Universal Robots PolyScope program: 0609.urp

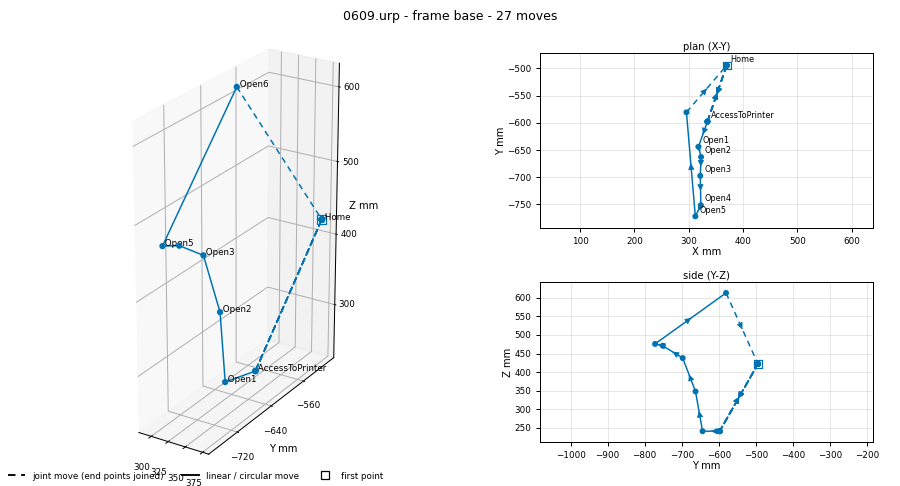
[picture p0: tool path of 0609.urp in frame base, 27 of 27 moves have a stored position in this frame; points joined in program order, loops and branches not executed]
Program 0609 (installation=default directory=/programs/usbdisk/새로운 폴더_2 createdIn=5.12.7.1102192 lastSavedIn=5.11.0.108249 robotSerialNumber=20215501208)
Calibrated DH parameters: a=[0.000135, -0.201821, -0.391913, -0.000063, 0.000038, 0]; d=[0.162484, -479.507804, 481.562221, -1.92078, 0.099549, 0.099572]; alpha=[1.570789, -0.00078, 0.007148, 1.569147, -1.569841, 0]; deltaTheta=[0, 1.075971, -1.038513, -0.037456, 0, 0]
Robot Program (runOnlyOnce=false)
  Folder Init
    Call Init_Variables
    Call Socket_Open
    MoveJ speed 60 deg/s, acceleration 80 deg/s^2 (useActiveTCP=true) feature=Base
      Waypoint Home: TCP in base x=369.65 y=-494.569 z=421.925 mm, rx=0.0496 ry=-3.0772 rz=-0.0574 rad; joints [-245.337, -73.512, 79.652, 267.34, -92.102, 23.034] deg
  Folder Main Sequence
    Folder Task1:OpenPrinter
      Call Enter_Next_Task
      Loop While (checkContinuously=false) expression=retry_count <= max_retry and task_done == 0
        MoveJ speed 60 deg/s, acceleration 80 deg/s^2 (useActiveTCP=true) feature=Base
          Waypoint Home: TCP in base x=369.65 y=-494.569 z=421.925 mm, rx=0.0496 ry=-3.0772 rz=-0.0574 rad; joints [-245.337, -73.512, 79.652, 267.34, -92.102, 23.034] deg
          Waypoint AccessToPrinter: TCP in base x=334.462 y=-597.737 z=240.467 mm, rx=-0.0069 ry=3.1388 rz=-0.0445 rad; joints [-252.013, -58.111, 86.313, 240.264, -90.06, 18.038] deg
          MoveL speed 250 mm/s, acceleration 1200 mm/s^2 (useActiveTCP=true) feature=Base
            Waypoint Open1: TCP in base x=318.021 y=-643.967 z=240.481 mm, rx=-0.0068 ry=3.1388 rz=-0.0445 rad; joints [-254.436, -54.011, 79.432, 243.032, -89.985, 15.598] deg
            Waypoint Open2: TCP in base x=322.784 y=-662.887 z=347.649 mm, rx=0.0033 ry=-3.1272 rz=-0.039 rad; joints [-254.437, -55.388, 64.401, 262.634, -90.038, 15.606] deg
            Waypoint Open3: TCP in base x=321.329 y=-697.509 z=437.722 mm, rx=0.0214 ry=3.1194 rz=-0.1204 rad; joints [-255.276, -52.597, 48.232, 269.856, -89.693, 15.609] deg
            Waypoint Open4: TCP in base x=322.369 y=-751.555 z=471.14 mm, rx=-0.056 ry=3.0495 rz=-0.4423 rad; joints [-256.148, -45.626, 35.019, 263.813, -89.938, 11.834] deg
            Waypoint Open5: TCP in base x=312.24 y=-772.06 z=475.94 mm, rx=-0.0354 ry=3.0161 rz=-0.6648 rad; joints [-256.943, -44.398, 34.822, 254.694, -91.917, 11.398] deg
            Waypoint Open6: TCP in base x=295.845 y=-580.619 z=613.456 mm, rx=-0.0405 ry=-3.057 rz=-0.0586 rad; joints [-254.175, -62.295, 34.865, 300.956, -93.656, 17.369] deg
        Call Check_Door_Open
        Switch expression=fail_flag
          Case (caseValue=0)
            Script: task_done = 1
          Case (caseValue=1)
            Script: retry_count = retry_count + 1
      If task_done == 0
        Call Error_Stop
    Folder Task2:PickA4FromTray
      Call Enter_Next_Task
      MoveJ speed 60 deg/s, acceleration 80 deg/s^2 (useActiveTCP=true) feature=Base
        Waypoint Home: TCP in base x=369.65 y=-494.569 z=421.925 mm, rx=0.0496 ry=-3.0772 rz=-0.0574 rad; joints [-245.337, -73.512, 79.652, 267.34, -92.102, 23.034] deg
        Waypoint AccessToTray: TCP in base x=369.603 y=-494.616 z=422.071 mm, rx=0.0496 ry=-3.0774 rz=-0.0569 rad; joints [-245.343, -73.517, 79.642, 267.335, -92.098, 23.025] deg
      Call Gripper_Open
      Call Wait_Motor_Idle
      Call DC_Run
      Call Wait_Motor_Idle
      Call Gripper_Close
      Call Wait_Motor_Idle
      MoveJ speed 60 deg/s, acceleration 80 deg/s^2 (useActiveTCP=true) feature=Base
        Waypoint RetreatFromTray: TCP in base x=369.611 y=-494.615 z=422.061 mm, rx=0.0496 ry=-3.0774 rz=-0.057 rad; joints [-245.343, -73.516, 79.642, 267.335, -92.097, 23.027] deg
      If fail_flag == 1
        Call Error_Stop
    Folder Task3:PlaceA4OnScanner
      Call Enter_Next_Task
      MoveJ speed 60 deg/s, acceleration 80 deg/s^2 (useActiveTCP=true) feature=Base
        Waypoint AccessToScanne: TCP in base x=369.631 y=-494.591 z=421.924 mm, rx=0.0495 ry=-3.0773 rz=-0.0574 rad; joints [-245.34, -73.511, 79.65, 267.341, -92.099, 23.034] deg
      Call Gripper_Open
      Call Wait_Motor_Idle
      MoveJ speed 60 deg/s, acceleration 80 deg/s^2 (useActiveTCP=true) feature=Base
        Waypoint RetreatFromScan: TCP in base x=369.639 y=-494.607 z=421.869 mm, rx=0.0495 ry=-3.0772 rz=-0.0575 rad; joints [-245.339, -73.506, 79.652, 267.339, -92.104, 23.035] deg
      Call Check_Paper_Detected
      If fail_flag == 1
        Call Error_Stop
    Folder Task4:ClosePrinter
      Call Enter_Next_Task
      Loop While (checkContinuously=false) expression=retry_count <= max_retry and task_done == 0
        MoveJ speed 60 deg/s, acceleration 80 deg/s^2 (useActiveTCP=true) feature=Base
          Waypoint AccessToPrinter: TCP in base x=334.462 y=-597.737 z=240.467 mm, rx=-0.0069 ry=3.1388 rz=-0.0445 rad; joints [-252.013, -58.111, 86.313, 240.264, -90.06, 18.038] deg
          Waypoint ClosePrinterr: TCP in base x=369.641 y=-494.609 z=421.879 mm, rx=0.0495 ry=-3.0772 rz=-0.0575 rad; joints [-245.339, -73.506, 79.651, 267.339, -92.101, 23.035] deg
          Waypoint RetreatFromPrin: TCP in base x=369.644 y=-494.592 z=421.887 mm, rx=0.0495 ry=-3.0772 rz=-0.0574 rad; joints [-245.338, -73.509, 79.653, 267.337, -92.102, 23.034] deg
        Call Check_Door_Closed
        Switch expression=fail_flag
          Case (caseValue=0)
            Script: task_done = 1
          Case (caseValue=1)
            Script: retry_count = retry_count + 1
      If task_done == 0
        Call Error_Stop
    Folder Task5:OpenPrinter
      Call Enter_Next_Task
      Loop While (checkContinuously=false) expression=retry_count <= max_retry and task_done == 0
        MoveJ speed 60 deg/s, acceleration 80 deg/s^2 (useActiveTCP=true) feature=Base
          Waypoint AccessToPrinter: TCP in base x=334.462 y=-597.737 z=240.467 mm, rx=-0.0069 ry=3.1388 rz=-0.0445 rad; joints [-252.013, -58.111, 86.313, 240.264, -90.06, 18.038] deg
          Waypoint OpenPrinterr: TCP in base x=369.668 y=-494.585 z=421.902 mm, rx=0.0496 ry=-3.0772 rz=-0.0574 rad; joints [-245.336, -73.508, 79.649, 267.341, -92.102, 23.034] deg
          Waypoint RetreatFromPrin: TCP in base x=369.644 y=-494.592 z=421.887 mm, rx=0.0495 ry=-3.0772 rz=-0.0574 rad; joints [-245.338, -73.509, 79.653, 267.337, -92.102, 23.034] deg
        Call Check_Door_Open
        Switch expression=fail_flag
          Case (caseValue=0)
            Script: task_done = 1
          Case (caseValue=1)
            Script: retry_count = retry_count + 1
      If task_done == 0
        Call Error_Stop
    Folder Task6:PickA4FromScanner
      Call Enter_Next_Task
      Call Gripper_Open
      Call Wait_Motor_Idle
      MoveJ speed 60 deg/s, acceleration 80 deg/s^2 (useActiveTCP=true) feature=Base
        Waypoint AccessToScanner: TCP in base x=369.655 y=-494.587 z=421.911 mm, rx=0.0495 ry=-3.0772 rz=-0.0574 rad; joints [-245.337, -73.508, 79.649, 267.341, -92.103, 23.036] deg
      Call Gripper_Close
      Call Wait_Motor_Idle
      MoveJ speed 60 deg/s, acceleration 80 deg/s^2 (useActiveTCP=true) feature=Base
        Waypoint RetreatFromSca: TCP in base x=369.664 y=-494.583 z=421.908 mm, rx=0.0496 ry=-3.0772 rz=-0.0574 rad; joints [-245.336, -73.508, 79.649, 267.341, -92.102, 23.034] deg
      If fail_flag == 1
        Call Error_Stop
    Folder Task7:PlaceA4InBasket
      Call Enter_Next_Task
      MoveJ speed 60 deg/s, acceleration 80 deg/s^2 (useActiveTCP=true) feature=Base
        Waypoint AccessToBasket: TCP in base x=369.638 y=-494.57 z=421.942 mm, rx=0.0496 ry=-3.0772 rz=-0.0573 rad; joints [-245.338, -73.513, 79.652, 267.339, -92.104, 23.032] deg
      Call Gripper_Open
      Call Wait_Motor_Idle
      MoveJ speed 60 deg/s, acceleration 80 deg/s^2 (useActiveTCP=true) feature=Base
        Waypoint RetreatFromBask: TCP in base x=369.654 y=-494.572 z=421.913 mm, rx=0.0496 ry=-3.0772 rz=-0.0574 rad; joints [-245.336, -73.511, 79.652, 267.339, -92.103, 23.033] deg
      If fail_flag == 1
        Call Error_Stop
    Folder Task8:ClosePrinter
      Call Enter_Next_Task
      Loop While (checkContinuously=false) expression=retry_count <= max_retry and task_done == 0
        MoveJ speed 60 deg/s, acceleration 80 deg/s^2 (useActiveTCP=true) feature=Base
          Waypoint AccessToPrinter: TCP in base x=334.462 y=-597.737 z=240.467 mm, rx=-0.0069 ry=3.1388 rz=-0.0445 rad; joints [-252.013, -58.111, 86.313, 240.264, -90.06, 18.038] deg
          Waypoint ClosePrinter: TCP in base x=369.674 y=-494.571 z=421.895 mm, rx=0.0496 ry=-3.0772 rz=-0.0574 rad; joints [-245.335, -73.508, 79.651, 267.341, -92.102, 23.034] deg
          Waypoint RetreatFromPrin: TCP in base x=369.644 y=-494.592 z=421.887 mm, rx=0.0495 ry=-3.0772 rz=-0.0574 rad; joints [-245.338, -73.509, 79.653, 267.337, -92.102, 23.034] deg
        Call Check_Door_Closed
        Switch expression=fail_flag
          Case (caseValue=0)
            Script: task_done = 1
          Case (caseValue=1)
            Script: retry_count = retry_count + 1
      If task_done == 0
        Call Error_Stop
SubProgram -> Socket_Open
SubProgram -> Init_Variables
SubProgram -> DC_Run
SubProgram -> Gripper_Close
SubProgram -> Gripper_Open
SubProgram -> Wait_Motor_Idle
SubProgram -> Check_Door_Closed
SubProgram -> Check_Door_Open
SubProgram -> Check_Paper_Detected
SubProgram -> Error_Stop
SubProgram -> Enter_Next_Task
SubProgram Init_Variables (keepSynchronizedWithDisk=false)
  Script file /programs/usbdisk/scripts/Init_Variables.script
    | # Retry / fail control
    | global retry_count = 0
    | global max_retry = 2
    | global fail_flag = 0
    | global task_done = 0
    | global current_task = 0
    | 
    | # State variables
    | global door_state = 0      # 0: closed, 1: open
    | global motor_state = 0     # 0: idle, 1: busy
    | global paper_state = 0     # 0: not detected, 1: detected
    | 
    | # Socket / response
    | global socket_state = False
    | global pc_response = ""
    | 
    | # ============================================================
    | # Command strings
    | # URScript → PC Server → Arduino
    | # ============================================================
    | 
    | global CMD_PING = "PING\n"
    | global CMD_GRIPPER_OPEN = "G OPEN\n"
    | global CMD_GRIPPER_CLOSE = "G CLOSE\n"
    | global CMD_DC_RUN = "D RUN\n"
    | global CMD_ESTOP = "ESTOP\n"
    | global CMD_MOTOR_STATUS = "MOTOR STATUS\n"
    | global CMD_DOOR_STATUS = "DOOR STATUS\n"
    | global CMD_CAMERA = "V CAMERA\n"
    | 
    | # ============================================================
    | # Expected response strings
    | # Arduino / PC Server → URScript
    | # ============================================================
    | 
    | global RESP_OK_PING = "OK PING"
    | global RESP_OK_GRIPPER_OPEN = "OK G OPEN"
    | global RESP_OK_GRIPPER_CLOSE = "OK G CLOSE"
    | global RESP_OK_DC_RUN = "OK D RUN"
    | global RESP_OK_ESTOP = "OK ESTOP"
    | 
    | global RESP_MOTOR_BUSY = "MOTOR STATUS BUSY"
    | global RESP_MOTOR_IDLE = "MOTOR STATUS IDLE"
    | 
    | global RESP_DOOR_OPEN = "DOOR STATUS OPEN"
    | global RESP_DOOR_CLOSED = "DOOR STATUS CLOSED"
    | 
    | global RESP_PAPER_DETECTED = "PAPER DETECTED"
    | global RESP_PAPER_NOT_DETECTED = "PAPER NOT DETECTED"
SubProgram Socket_Open (keepSynchronizedWithDisk=false)
  Script file /programs/usbdisk/scripts/Socket_Open.script
    | global socket_state = socket_open("192.168.0.10", 5000)
    | 
    | if socket_state:
    |   socket_send_string(CMD_PING)
    |   global pc_response = socket_read_line()
    | 
    |   if pc_response == RESP_OK_PING:
    |     global fail_flag = 0
    |     textmsg("Socket open OK")
    |   else:
    |     global fail_flag = 1
    |     textmsg("PING failed: ", pc_response)
    |   end
    | 
    | else:
    |   global fail_flag = 1
    |   textmsg("Socket open FAILED")
    |   halt
    | end
SubProgram Enter_Next_Task (keepSynchronizedWithDisk=false)
  Script file /programs/usbdisk/scripts/Enter_Next_Task.script
    | global current_task = current_task + 1
    | global retry_count = 0
    | global task_done = 0
    | global fail_flag = 0
SubProgram Check_Door_Open (keepSynchronizedWithDisk=false)
  Script file /programs/usbdisk/Check_Door_Open.script
    | socket_send_string(CMD_DOOR_STATUS)
    | global pc_response = socket_read_line()
    | 
    | if pc_response == RESP_DOOR_OPEN:
    |   global door_state = 1
    |   global fail_flag = 0
    | 
    | elif pc_response == RESP_DOOR_CLOSED:
    |   global door_state = 0
    |   global fail_flag = 1
    | 
    | else:
    |   global fail_flag = 1
    | end
SubProgram Error_Stop (keepSynchronizedWithDisk=false)
  Script file /programs/usbdisk/Error_Stop.script
    | # 현재 task 번호에 따라 오류 메시지 출력
    | if current_task == 1:
    |   popup("Task 1 Failed: Open Printer", title="Task Error", warning=True, error=False)
    | 
    | elif current_task == 2:
    |   popup("Task 2 Failed: Pick A4 From Paper Box", title="Task Error", warning=True, error=False)
    | 
    | elif current_task == 3:
    |   popup("Task 3 Failed: Place A4 To Printer Head", title="Task Error", warning=True, error=False)
    | 
    | elif current_task == 4:
    |   popup("Task 4 Failed: Close Printer", title="Task Error", warning=True, error=False)
    | 
    | elif current_task == 5:
    |   popup("Task 5 Failed: Open Printer Again", title="Task Error", warning=True, error=False)
    | 
    | elif current_task == 6:
    |   popup("Task 6 Failed: Pick A4 From Printer Head", title="Task Error", warning=True, error=False)
    | 
    | elif current_task == 7:
    |   popup("Task 7 Failed: Place A4 To Paper Box", title="Task Error", warning=True, error=False)
    | 
    | elif current_task == 8:
    |   popup("Task 8 Failed: Close Printer Again", title="Task Error", warning=True, error=False)
    | 
    | else:
    |   popup("Unknown Task Failed", title="Task Error", warning=True, error=False)
    | end
    | 
    | # Arduino/PC 측 정지 요청
    | socket_send_string(CMD_ESTOP)
    | global pc_response = socket_read_line()
    | 
    | # 로그 출력
    | textmsg("ESTOP response: ", pc_response)
    | 
    | # UR Program 정지
    | halt
SubProgram Gripper_Open (keepSynchronizedWithDisk=false)
  Script file /programs/usbdisk/Gripper_Open.script
    | socket_send_string(CMD_GRIPPER_OPEN)
    | global pc_response = socket_read_line()
    | 
    | if pc_response == RESP_OK_GRIPPER_OPEN:
    |   global motor_state = 1
    |   global fail_flag = 0
    | else:
    |   global fail_flag = 1
    | end
SubProgram Wait_Motor_Idle (keepSynchronizedWithDisk=false)
  Script file /programs/usbdisk/scripts/Wait_Motor_Idle.script
    | # MOTOR STATUS를 반복 조회하여 IDLE이 될 때까지 대기
    | # break문 사용 불가하므로 wait_done 임시 변수 사용
    | 
    | wait_done = 0
    | 
    | while wait_done == 0:
    |   socket_send_string(CMD_MOTOR_STATUS)
    |   global pc_response = socket_read_line()
    | 
    |   if pc_response == RESP_MOTOR_BUSY:
    |     global motor_state = 1
    |     sleep(0.1)
    | 
    |   elif pc_response == RESP_MOTOR_IDLE:
    |     global motor_state = 0
    |     global fail_flag = 0
    |     global wait_done = 1
    | 
    |   else:
    |     global fail_flag = 1
    |     global wait_done = 1
    |   end
    | end
SubProgram DC_Run (keepSynchronizedWithDisk=false)
  Script file /programs/usbdisk/DC_Run.script
    | socket_send_string(CMD_DC_RUN)
    | global pc_response = socket_read_line()
    | 
    | if pc_response == RESP_OK_DC_RUN:
    |   global motor_state = 1
    |   global fail_flag = 0
    | else:
    |   global fail_flag = 1
    | end
SubProgram Gripper_Close (keepSynchronizedWithDisk=false)
  Script file /programs/usbdisk/scripts/Gripper_Close.script
    | socket_send_string(CMD_GRIPPER_CLOSE)
    | global pc_response = socket_read_line()
    | 
    | if pc_response == RESP_OK_GRIPPER_CLOSE:
    |   global motor_state = 1
    |   global fail_flag = 0
    | else:
    |   global fail_flag = 1
    | end
SubProgram Check_Paper_Detected (keepSynchronizedWithDisk=false)
  Script file /programs/usbdisk/scripts/Check_Paper_Detected.script
    | socket_send_string(CMD_CAMERA)
    | global pc_response = socket_read_line()
    | 
    | if pc_response == RESP_PAPER_DETECTED:
    |   global paper_state = 1
    |   global fail_flag = 0
    | 
    | elif pc_response == RESP_PAPER_NOT_DETECTED:
    |   global paper_state = 0
    |   global fail_flag = 1
    | 
    | else:
    |   global fail_flag = 1
    | end
SubProgram Check_Door_Closed (keepSynchronizedWithDisk=false)
  Script file /programs/usbdisk/Check_Door_Closed.script
    | socket_send_string(CMD_DOOR_STATUS)
    | global pc_response = socket_read_line()
    | 
    | if pc_response == RESP_DOOR_CLOSED:
    |   global door_state = 0
    |   global fail_flag = 0
    | 
    | elif pc_response == RESP_DOOR_OPEN:
    |   global door_state = 1
    |   global fail_flag = 1
    | 
    | else:
    |   global fail_flag = 1
    | end
